// TIA Portal project "EM1-2-Basisinstructies en timers_V15.1" (V15.1)

(* hardware
DEVICE "S7-1200 station_1"  S7-1200 Station
   slot 0: "Rack_0"  S7-1200 Rack  Rack  V1.0
   slot 1: "PLC_1"  CPU 1214C AC/DC/Rly  6ES7 214-1BG31-0XB0  V3.0
   slot 2: "DI 8x24VDC_1"  SM 1221 DI8 x 24VDC  6ES7 221-1BF30-0XB0  V1.0
   slot 3: "AQ 1x12BIT_1"  AQ1 signal board  6ES7 232-4HA30-0XB0  V1.0
*)

// ===== PLC "PLC_1"  CPU 1214C AC/DC/Rly =====

VAR_GLOBAL   // PLC tag table "Default tag table"
   "mSystem_Byte" AT %MB254 : Byte;   // System byte
   "mFirstScan" AT %M254.0 : Bool;   // Bit only TRUE during the first scan
   "mDiagStatusUpdate" AT %M254.1 : Bool;   // New diagnostic status available
   "mAlwaysTRUE" AT %M254.2 : Bool;   // Bit always TRUE
   "mAlwaysFALSE" AT %M254.3 : Bool;   // Bit always FALSE
   "mClock_Byte" AT %MB255 : Byte;   // Clock memory byte
   "mClock_10Hz" AT %M255.0 : Bool;   // Clock memory bit - 10 Hz
   "mClock_5Hz" AT %M255.1 : Bool;   // Clock memory bit - 5 Hz
   "mClock_2.5Hz" AT %M255.2 : Bool;   // Clock memory bit - 2.5 Hz
   "mClock_2Hz" AT %M255.3 : Bool;   // Clock memory bit - 2 Hz
   "mClock_1.25Hz" AT %M255.4 : Bool;   // Clock memory bit - 1.25 Hz
   "mClock_1Hz" AT %M255.5 : Bool;   // Clock memory bit - 1 Hz
   "mClock_0.625Hz" AT %M255.6 : Bool;   // Clock memory bit - 0.625 Hz
   "mClock_0.5Hz" AT %M255.7 : Bool;   // Clock memory bit - 0.5 Hz
END_VAR

VAR_GLOBAL   // PLC tag table "Table_IO"
   "iSelEmergency-S5" AT %I0.4 : Bool;   // Sewitch emergency operation
   "oS1_LmpGreen_H1" AT %Q0.0 : Bool;   // Traffic sign 1 – Green light
   "oS2_LmpGreen_H2" AT %Q0.1 : Bool;   // Traffic sign 2 – Green light
   "oS1_LmpOrange_H3" AT %Q0.2 : Bool;   // Traffic sign 1 – Orange light
   "oS1_LmpRed_H5" AT %Q0.4 : Bool;   // Traffic sign 1 – Red light
   "oS2-LmpRed_H6" AT %Q0.5 : Bool;   // Traffic sign 2 – Red light
   "oS2_LmpOrange_H4" AT %Q0.3 : Bool;   // Traffic sign 2 – Orange light
   "oRelFreezeError" AT %Q1.0 : Bool;   // Freeze error relay
END_VAR

VAR_GLOBAL   // PLC tag table "Table_Flags"
   "mFrom1to2" AT %M0.0 : Bool;   // Traffic from sign 1 to 2
   "mWarning1to2" AT %M0.1 : Bool;   // Warning traffic on sign 1
   "mFrom2to1" AT %M0.2 : Bool;   // Traffic from sign 2 to 1
   "mWarning2to1" AT %M0.3 : Bool;   // Warning traffic on sign 2
   "mpfSelEmergency_S5" AT %M2.0 : Bool;   // Rising edge iSelEmergency_S5
   "mNormalByte" AT %MB0 : Byte;   // Normal functionality byte
   "mPrevNormalByte" AT %MB1 : Byte;   // Previous status of mNormalByte
END_VAR

// folder: System blocks/Program resources

DATA_BLOCK "DB_TON1"   // DB1
{ S7_Optimized_Access := 'TRUE' }
AUTHOR : Simatic
FAMILY : IEC
NAME : IEC_TMR
VERSION : 1.0
// stored: InstanceOfName IEC_TIMER
"IEC_TIMER"
BEGIN
END_DATA_BLOCK

DATA_BLOCK "DB_TON2"   // DB2
{ S7_Optimized_Access := 'TRUE' }
AUTHOR : Simatic
FAMILY : IEC
NAME : IEC_TMR
VERSION : 1.0
// stored: InstanceOfName IEC_TIMER
"IEC_TIMER"
BEGIN
END_DATA_BLOCK

DATA_BLOCK "DB_TON3"   // DB3
{ S7_Optimized_Access := 'TRUE' }
AUTHOR : Simatic
FAMILY : IEC
NAME : IEC_TMR
VERSION : 1.0
// stored: InstanceOfName IEC_TIMER
"IEC_TIMER"
BEGIN
END_DATA_BLOCK

DATA_BLOCK "IEC_TON1"   // DB4
{ S7_Optimized_Access := 'TRUE' }
AUTHOR : Simatic
FAMILY : IEC
NAME : IEC_TMR
VERSION : 1.0
// stored: InstanceOfName IEC_TIMER
"IEC_TIMER"
BEGIN
END_DATA_BLOCK

// folder: (top level)

FUNCTION "FC_Sign1" : Void   // FC1, FBD
TITLE = Sign 1
{ S7_Optimized_Access := 'TRUE' }
VERSION : 0.1
BEGIN

REGION Network 1: Red lamp - STOP
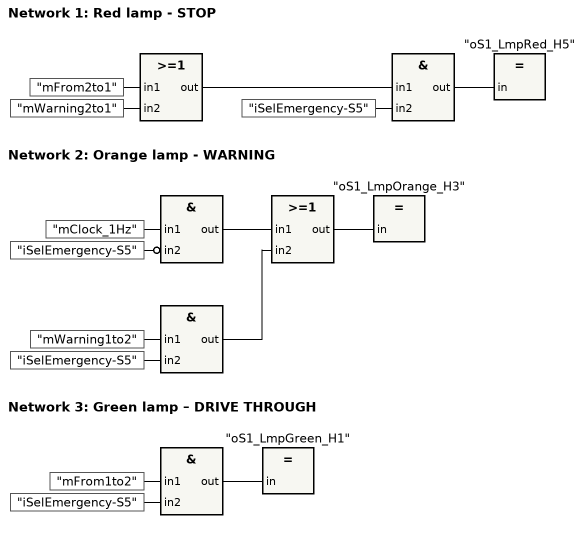
   "oS1_LmpRed_H5" := ("mFrom2to1" OR "mWarning2to1") AND "iSelEmergency-S5";
END_REGION

REGION Network 2: Orange lamp - WARNING
   // - Indien de schakelaar “iSelFout-S5” de status FALSE heeft moet de oranje waarschuwingslamp knipperen met een frequentie van 1 Hz.
   // - Indien de schakelaar “iSelFout-S5” de status TRUE heeft moet de oranje waarschuwingslamp continue branden indien de variabele “mOpgelet1naar2” de status TRUE heeft
   "oS1_LmpOrange_H3" := ("mClock_1Hz" AND NOT "iSelEmergency-S5") OR ("mWarning1to2" AND "iSelEmergency-S5");
END_REGION

REGION Network 3: Green lamp – DRIVE THROUGH
   "oS1_LmpGreen_H1" := "mFrom1to2" AND "iSelEmergency-S5";
END_REGION
END_FUNCTION

FUNCTION "FC_Sign2" : Void   // FC2, LAD
TITLE = Sign 2
{ S7_Optimized_Access := 'TRUE' }
VERSION : 0.1
BEGIN

REGION Network 1: Red lamp - STOP
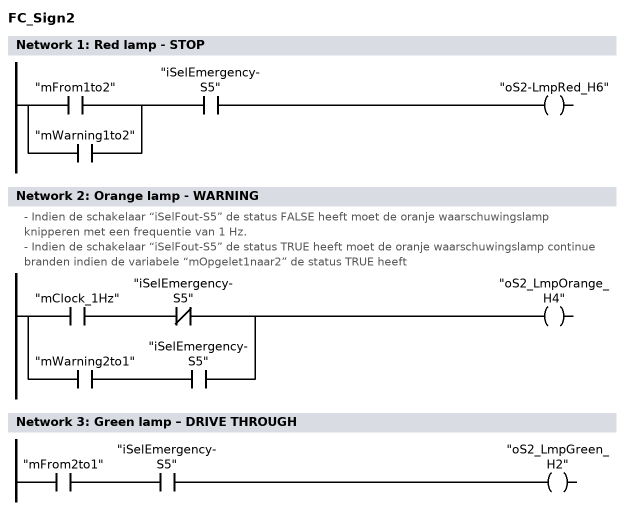
   RUNG wire#powerrail
      Contact( "mFrom1to2" )
      wire#w1
      Contact( "iSelEmergency-S5" )
      Coil( "oS2-LmpRed_H6" )
   END_RUNG
   RUNG wire#powerrail
      Contact( "mWarning1to2" )
   END_RUNG wire#w1
   // the same network as SCL:
   "oS2-LmpRed_H6" := ("mFrom1to2" OR "mWarning1to2") AND "iSelEmergency-S5";
END_REGION

REGION Network 2: Orange lamp - WARNING
   // - Indien de schakelaar “iSelFout-S5” de status FALSE heeft moet de oranje waarschuwingslamp knipperen met een frequentie van 1 Hz.
   // - Indien de schakelaar “iSelFout-S5” de status TRUE heeft moet de oranje waarschuwingslamp continue branden indien de variabele “mOpgelet1naar2” de status TRUE heeft
   RUNG wire#powerrail
      Contact( "mClock_1Hz" )
      I_Contact( "iSelEmergency-S5" )
      wire#w1
      Coil( "oS2_LmpOrange_H4" )
   END_RUNG
   RUNG wire#powerrail
      Contact( "mWarning2to1" )
      Contact( "iSelEmergency-S5" )
   END_RUNG wire#w1
   // the same network as SCL:
   "oS2_LmpOrange_H4" := ("mClock_1Hz" AND NOT "iSelEmergency-S5") OR ("mWarning2to1" AND "iSelEmergency-S5");
END_REGION

REGION Network 3: Green lamp – DRIVE THROUGH
   RUNG wire#powerrail
      Contact( "mFrom2to1" )
      Contact( "iSelEmergency-S5" )
      Coil( "oS2_LmpGreen_H2" )
   END_RUNG
   // the same network as SCL:
   "oS2_LmpGreen_H2" := "mFrom2to1" AND "iSelEmergency-S5";
END_REGION
END_FUNCTION

FUNCTION "FC_Normal" : Void   // FC3, FBD
TITLE = Normal operation
{ S7_Optimized_Access := 'TRUE' }
VERSION : 0.1
   VAR_TEMP   // added for the SCL form of the ladder/FBD networks
      _w1 : Bool;
   END_VAR
BEGIN

REGION Network 1: Activate normal operation
   // Change the state of the next PLC TAGs when switching the selector switch “iSelEmergency_S5” from status FALSE to TRUE: 
   // -   mFrom1to2       TRUE
   // -   mWarning1to2  FALSE 
   // -   mFrom2to1       FALSE 
   // -   mWarning2to1  FALSE
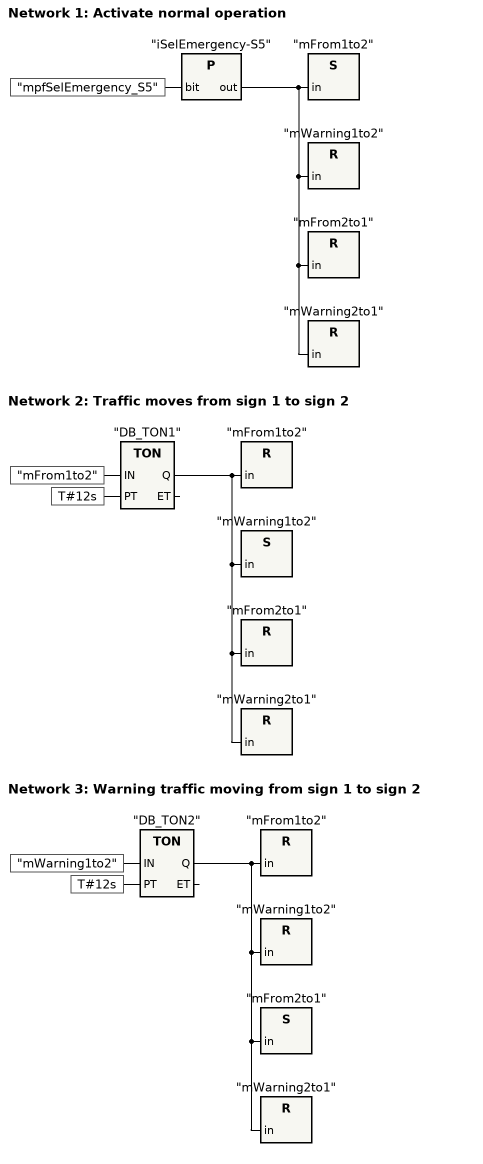
   #_w1 := "iSelEmergency-S5" AND NOT "mpfSelEmergency_S5";   // rising edge of "iSelEmergency-S5"
   "mpfSelEmergency_S5" := "iSelEmergency-S5";
   IF #_w1 THEN
       "mFrom1to2" := TRUE;
       "mWarning1to2" := FALSE;
       "mFrom2to1" := FALSE;
       "mWarning2to1" := FALSE;
   END_IF;
END_REGION

REGION Network 2: Traffic moves from sign 1 to sign 2
   // Traffic is allowed for 12 s to move from traffic sign 1 to traffic sign 2. Status of the PLC TAGS during these 12 s: 
   // -   mFrom1to2       TRUE
   // -   mWarning1to2  FALSE 
   // -   mFrom2to1       FALSE 
   // -   mWarning2to1  FALSE 
   // 
   // After these 12 s the state of the PLC TAGs change to: 
   // -   mFrom1to2       FALSE 
   // -   mWarning1to2  TRUE
   // -   mFrom2to1       FALSE 
   // -   mWarning2to1  FALSE
   "DB_TON1".TON(IN := "mFrom1to2", PT := T#12s);
   IF "DB_TON1".Q THEN
       "mFrom1to2" := FALSE;
       "mWarning1to2" := TRUE;
       "mFrom2to1" := FALSE;
       "mWarning2to1" := FALSE;
   END_IF;
END_REGION

REGION Network 3: Warning traffic moving from sign 1 to sign 2
   // The orange lamp warns the traffic for a change of direction during 3 s  at traffic sign 1. Status of the PLC TAGS during these 3 s: 
   // -   mFrom1to2        FALSE 
   // -   mWarning1to2  TRUE
   // -   mFrom2to1        FALSE 
   // -   mWarning2to1   FALSE 
   // 
   // After these 3 s the state of the PLC TAGs change to: 
   // -   mFrom1to2       FALSE 
   // -   mWarning1to2  FALSE 
   // -   mFrom2to1       TRUE
   // -   mWarning2to1  FALSE
   "DB_TON2".TON(IN := "mWarning1to2", PT := T#12s);
   IF "DB_TON2".Q THEN
       "mFrom1to2" := FALSE;
       "mWarning1to2" := FALSE;
       "mFrom2to1" := TRUE;
       "mWarning2to1" := FALSE;
   END_IF;
END_REGION

REGION Network 4: Traffic moves from sign 2 to sign 1
   // Traffic is allowed for 12 s to move from traffic sign 2 to traffic sign 1. Status of the PLC TAGS during these 12 s: 
   // -   mFrom1to2       FALSE 
   // -   mWarning1to2  FALSE 
   // -   mFrom2to1       TRUE
   // -   mWarning2to1  FALSE 
   // 
   // After these 12 s the state of the PLC TAGs change to: 
   // -   mFrom1to2       FALSE 
   // -   mWarning1to2  FALSE 
   // -   mFrom2to1       FALSE 
   // -   mWarning2to1  TRUE
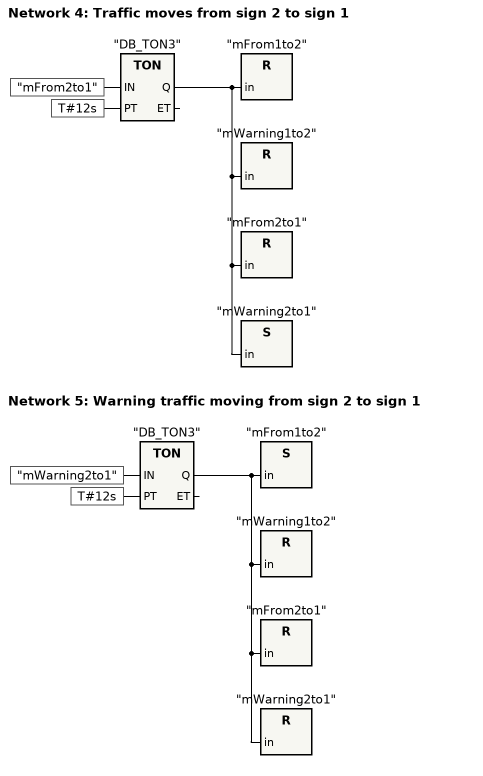
   "DB_TON3".TON(IN := "mFrom2to1", PT := T#12s);
   IF "DB_TON3".Q THEN
       "mFrom1to2" := FALSE;
       "mWarning1to2" := FALSE;
       "mFrom2to1" := FALSE;
       "mWarning2to1" := TRUE;
   END_IF;
END_REGION

REGION Network 5: Warning traffic moving from sign 2 to sign 1
   // The orange lamp warns the traffic for a change of direction during 3 s  at traffic sign 2. Status of the PLC TAGS during these 3 s: 
   // -   mFrom1to2       FALSE 
   // -   mWarning1to2  FALSE 
   // -   mFrom2to1       FALSE 
   // -   mWarning2to1  TRUE
   // 
   // After these 3 s the state of the PLC TAGs change to (which is the same situation as in network 2): 
   // -   mFrom1to2       TRUE
   // -   mWarning1to2  FALSE 
   // -   mFrom2to1       FALSE 
   // -   mWarning2to1  FALSE
   "DB_TON3".TON(IN := "mWarning2to1", PT := T#12s);
   IF "DB_TON3".Q THEN
       "mFrom1to2" := TRUE;
       "mWarning1to2" := FALSE;
       "mFrom2to1" := FALSE;
       "mWarning2to1" := FALSE;
   END_IF;
END_REGION
END_FUNCTION

FUNCTION "FC_FreezeError" : Void   // FC4, SCL
{ S7_Optimized_Access := 'TRUE' }
VERSION : 0.1
BEGIN
   //TON Timer
   "IEC_TON1".TON(IN:=( "mNormalByte" = "mPrevNormalByte") AND "iSelEmergency-S5"=TRUE,
                  PT:=T#30s);

   //IF .. THEN .. ELSE
   IF "IEC_TON1".Q = TRUE THEN
       //Activate Freeze Error ouput
       "oRelFreezeError":=TRUE;
   ELSE
       //Deactivate Freeze Error ouput
       "oRelFreezeError":=FALSE;
   END_IF;

   //Make previous value of byte
   "mPrevNormalByte" := "mNormalByte";
END_FUNCTION

ORGANIZATION_BLOCK "Main"   // OB1, FBD, ProgramCycle
TITLE = "Main Program Sweep (Cycle)"
{ S7_Optimized_Access := 'TRUE' }
VERSION : 0.1
BEGIN

REGION Network 1: Normal operation
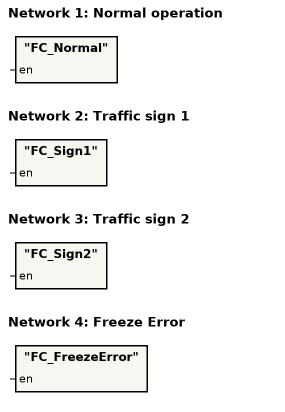
   "FC_Normal"();
END_REGION

REGION Network 2: Traffic sign 1
   "FC_Sign1"();
END_REGION

REGION Network 3: Traffic sign 2
   "FC_Sign2"();
END_REGION

REGION Network 4: Freeze Error
   "FC_FreezeError"();
END_REGION
END_ORGANIZATION_BLOCK